FUNCTION_BLOCK MOD_StateLogic (* PackML module state machine: commands only from the occupation owner and only where PackML allows them; runs the Resetting and Stopping procedures; Stopping waits until no skill is active *)
  (* Standard: 61499-2 *)
  (* Version 0.1, 2026-09-28, Project contributors, AAU Smart Production Lab *)
  PACKAGE modlib;
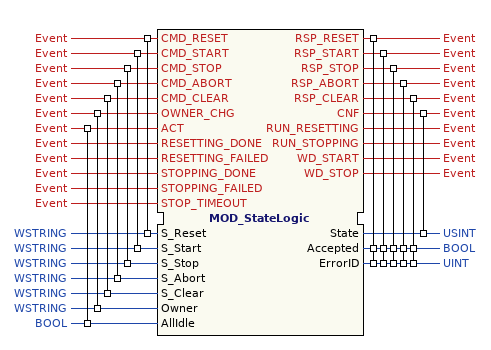
  EVENT_INPUT
    CMD_RESET WITH S_Reset;
    CMD_START WITH S_Start;
    CMD_STOP WITH S_Stop;
    CMD_ABORT WITH S_Abort;
    CMD_CLEAR WITH S_Clear;
    OWNER_CHG WITH Owner;
    ACT WITH AllIdle;
    RESETTING_DONE;
    RESETTING_FAILED;
    STOPPING_DONE;
    STOPPING_FAILED;
    STOP_TIMEOUT;
  END_EVENT
  EVENT_OUTPUT
    RSP_RESET WITH Accepted, ErrorID;
    RSP_START WITH Accepted, ErrorID;
    RSP_STOP WITH Accepted, ErrorID;
    RSP_ABORT WITH Accepted, ErrorID;
    RSP_CLEAR WITH Accepted, ErrorID;
    CNF WITH State;
    RUN_RESETTING;
    RUN_STOPPING;
    WD_START;
    WD_STOP;
  END_EVENT
  VAR_INPUT
    S_Reset : WSTRING;
    S_Start : WSTRING;
    S_Stop : WSTRING;
    S_Abort : WSTRING;
    S_Clear : WSTRING;
    Owner : WSTRING;
    AllIdle : BOOL := TRUE;
  END_VAR
  VAR_OUTPUT
    State : USINT := 2;
    Accepted : BOOL;
    ErrorID : UINT;
  END_VAR
  VAR
    Owned : BOOL;
    Here : USINT;
  END_VAR
  EC_STATES
    Stopped : Alg_Stopped -> CNF;
    Resetting : Alg_Resetting -> CNF, -> RUN_RESETTING;
    ResettingW : Alg_ResettingW;
    Idle : Alg_Idle -> CNF;
    Starting : Alg_Starting -> CNF;
    Execute : Alg_Execute -> CNF;
    Stopping : Alg_Stopping -> CNF, -> WD_START;
    StoppingW : Alg_StoppingW;
    StopProc : -> WD_STOP, -> RUN_STOPPING;
    StopProcW : Alg_StopProcW;
    Aborting : Alg_Aborting -> CNF, -> WD_STOP;
    Aborted : Alg_Aborted -> CNF;
    Clearing : Alg_Clearing -> CNF;
    ChkReset : Alg_ChkReset -> RSP_RESET;
    ChkStart : Alg_ChkStart -> RSP_START;
    ChkStop : Alg_ChkStop -> RSP_STOP;
    ChkAbort : Alg_ChkAbort -> RSP_ABORT;
    ChkClear : Alg_ChkClear -> RSP_CLEAR;
  END_STATES
  EC_TRANSITIONS
    Stopped TO ChkReset := CMD_RESET;
    ResettingW TO ChkReset := CMD_RESET;
    Idle TO ChkReset := CMD_RESET;
    Execute TO ChkReset := CMD_RESET;
    StoppingW TO ChkReset := CMD_RESET;
    StopProcW TO ChkReset := CMD_RESET;
    Aborted TO ChkReset := CMD_RESET;
    ChkReset TO Resetting := Accepted;
    ChkReset TO Stopped := Here = 0;
    ChkReset TO ResettingW := Here = 1;
    ChkReset TO Idle := Here = 2;
    ChkReset TO Execute := Here = 3;
    ChkReset TO StoppingW := Here = 4;
    ChkReset TO StopProcW := Here = 5;
    ChkReset TO Aborted := Here = 6;
    Stopped TO ChkStart := CMD_START;
    ResettingW TO ChkStart := CMD_START;
    Idle TO ChkStart := CMD_START;
    Execute TO ChkStart := CMD_START;
    StoppingW TO ChkStart := CMD_START;
    StopProcW TO ChkStart := CMD_START;
    Aborted TO ChkStart := CMD_START;
    ChkStart TO Starting := Accepted;
    ChkStart TO Stopped := Here = 0;
    ChkStart TO ResettingW := Here = 1;
    ChkStart TO Idle := Here = 2;
    ChkStart TO Execute := Here = 3;
    ChkStart TO StoppingW := Here = 4;
    ChkStart TO StopProcW := Here = 5;
    ChkStart TO Aborted := Here = 6;
    Stopped TO ChkStop := CMD_STOP;
    ResettingW TO ChkStop := CMD_STOP;
    Idle TO ChkStop := CMD_STOP;
    Execute TO ChkStop := CMD_STOP;
    StoppingW TO ChkStop := CMD_STOP;
    StopProcW TO ChkStop := CMD_STOP;
    Aborted TO ChkStop := CMD_STOP;
    ChkStop TO Stopping := Accepted;
    ChkStop TO Stopped := Here = 0;
    ChkStop TO ResettingW := Here = 1;
    ChkStop TO Idle := Here = 2;
    ChkStop TO Execute := Here = 3;
    ChkStop TO StoppingW := Here = 4;
    ChkStop TO StopProcW := Here = 5;
    ChkStop TO Aborted := Here = 6;
    Stopped TO ChkAbort := CMD_ABORT;
    ResettingW TO ChkAbort := CMD_ABORT;
    Idle TO ChkAbort := CMD_ABORT;
    Execute TO ChkAbort := CMD_ABORT;
    StoppingW TO ChkAbort := CMD_ABORT;
    StopProcW TO ChkAbort := CMD_ABORT;
    Aborted TO ChkAbort := CMD_ABORT;
    ChkAbort TO Aborting := Accepted;
    ChkAbort TO Stopped := Here = 0;
    ChkAbort TO ResettingW := Here = 1;
    ChkAbort TO Idle := Here = 2;
    ChkAbort TO Execute := Here = 3;
    ChkAbort TO StoppingW := Here = 4;
    ChkAbort TO StopProcW := Here = 5;
    ChkAbort TO Aborted := Here = 6;
    Stopped TO ChkClear := CMD_CLEAR;
    ResettingW TO ChkClear := CMD_CLEAR;
    Idle TO ChkClear := CMD_CLEAR;
    Execute TO ChkClear := CMD_CLEAR;
    StoppingW TO ChkClear := CMD_CLEAR;
    StopProcW TO ChkClear := CMD_CLEAR;
    Aborted TO ChkClear := CMD_CLEAR;
    ChkClear TO Clearing := Accepted;
    ChkClear TO Stopped := Here = 0;
    ChkClear TO ResettingW := Here = 1;
    ChkClear TO Idle := Here = 2;
    ChkClear TO Execute := Here = 3;
    ChkClear TO StoppingW := Here = 4;
    ChkClear TO StopProcW := Here = 5;
    ChkClear TO Aborted := Here = 6;
    Resetting TO ResettingW := 1;
    ResettingW TO Idle := RESETTING_DONE;
    ResettingW TO Aborting := RESETTING_FAILED;
    Starting TO Execute := 1;
    Stopping TO StoppingW := 1;
    StoppingW TO StopProc := AllIdle;
    StoppingW TO Aborting := STOP_TIMEOUT;
    StopProc TO StopProcW := 1;
    StopProcW TO Stopped := STOPPING_DONE;
    StopProcW TO Aborting := STOPPING_FAILED;
    Aborting TO Aborted := 1;
    Clearing TO Stopped := 1;
  END_TRANSITIONS
  ALGORITHM Alg_Stopped IN ST:
State := 2;
Here := 0;
  END_ALGORITHM
  ALGORITHM Alg_Resetting IN ST:
State := 15;
  END_ALGORITHM
  ALGORITHM Alg_ResettingW IN ST:
Here := 1;
  END_ALGORITHM
  ALGORITHM Alg_Idle IN ST:
State := 4;
Here := 2;
  END_ALGORITHM
  ALGORITHM Alg_Starting IN ST:
State := 3;
  END_ALGORITHM
  ALGORITHM Alg_Execute IN ST:
State := 6;
Here := 3;
  END_ALGORITHM
  ALGORITHM Alg_Stopping IN ST:
State := 7;
  END_ALGORITHM
  ALGORITHM Alg_StoppingW IN ST:
Here := 4;
  END_ALGORITHM
  ALGORITHM Alg_StopProcW IN ST:
Here := 5;
  END_ALGORITHM
  ALGORITHM Alg_Aborting IN ST:
State := 8;
  END_ALGORITHM
  ALGORITHM Alg_Aborted IN ST:
State := 9;
Here := 6;
  END_ALGORITHM
  ALGORITHM Alg_Clearing IN ST:
State := 1;
  END_ALGORITHM
  ALGORITHM Alg_ChkReset IN ST:
Owned := (S_Reset = Owner) AND (Owner <> "");
Accepted := Owned AND ((Here = 0));
IF NOT Owned THEN
  ErrorID := 5;
ELSIF NOT Accepted THEN
  ErrorID := 4;
ELSE
  ErrorID := 0;
END_IF;
  END_ALGORITHM
  ALGORITHM Alg_ChkStart IN ST:
Owned := (S_Start = Owner) AND (Owner <> "");
Accepted := Owned AND ((Here = 2));
IF NOT Owned THEN
  ErrorID := 5;
ELSIF NOT Accepted THEN
  ErrorID := 4;
ELSE
  ErrorID := 0;
END_IF;
  END_ALGORITHM
  ALGORITHM Alg_ChkStop IN ST:
Owned := (S_Stop = Owner) AND (Owner <> "");
Accepted := Owned AND ((Here = 1) OR (Here = 2) OR (Here = 3));
IF NOT Owned THEN
  ErrorID := 5;
ELSIF NOT Accepted THEN
  ErrorID := 4;
ELSE
  ErrorID := 0;
END_IF;
  END_ALGORITHM
  ALGORITHM Alg_ChkAbort IN ST:
Owned := (S_Abort = Owner) AND (Owner <> "");
Accepted := Owned AND ((Here = 0) OR (Here = 1) OR (Here = 2) OR (Here = 3) OR (Here = 4) OR (Here = 5));
IF NOT Owned THEN
  ErrorID := 5;
ELSIF NOT Accepted THEN
  ErrorID := 4;
ELSE
  ErrorID := 0;
END_IF;
  END_ALGORITHM
  ALGORITHM Alg_ChkClear IN ST:
Owned := (S_Clear = Owner) AND (Owner <> "");
Accepted := Owned AND ((Here = 6));
IF NOT Owned THEN
  ErrorID := 5;
ELSIF NOT Accepted THEN
  ErrorID := 4;
ELSE
  ErrorID := 0;
END_IF;
  END_ALGORITHM
END_FUNCTION_BLOCK
